(* IEC 61131-3 sources: Industry-PLC-LLM/data/PLCBEAD_repo/PLCBEAD_PLCEmbed-main/PLC-BEAD/Source/GEB/SEL2_OF_3B, 1 file *)

(* ---- SEL2_OF_3B.ST ---- *)
FUNCTION_BLOCK SEL2_OF_3B_Block

	VAR_INPUT
		IN1 :	BOOL;
		IN2 :	BOOL;
		IN3 :	BOOL;
		TD :	TIME;
	END_VAR

	VAR_OUTPUT
		Q :	BOOL;
		W :	BOOL;
	END_VAR

	VAR
		TDEL :	TON;
	END_VAR

	Q := (IN1 AND IN2) OR (IN1 AND IN3) OR (IN2 AND IN3);
	TDEL(IN := (IN1 XOR IN2) OR (IN1 XOR IN3) OR (IN2 XOR IN3), PT := TD);
	W := TDEL.Q;

END_FUNCTION_BLOCK

PROGRAM program0

	VAR
		IN1 :	BOOL;
		IN2 :	BOOL;
		IN3 :	BOOL;
		TD :	TIME;
		Q :	BOOL;
		W :	BOOL;
		func_block : SEL2_OF_3B_Block;
  	END_VAR
	func_block.IN1  :=IN1;
	func_block.IN2  :=IN2;
	func_block.IN3  :=IN3;
	func_block.TD  :=TD;
	func_block();
	Q := func_block.Q;
	W := func_block.W;

END_PROGRAM
